TEXTLIST PanelCmbTxtList
  1 = '1'
  2 = '2'
  3 = '3'
  4 = '4'
   = ''
END_TEXTLIST

(* stored: Version 1.1.0.1, ProductVersion 3.1.4024.4
   TextList PanelCmbTxtList: Id {5339c4ed-a166-42e8-a33c-cb84562f31b3} *)
